// TIA Portal V20 export
TYPE "LConSMC_typeLineAxisActValues"
// Istwerte der Bahn / Actuak values of the web
// stored: Access Published
   STRUCT
      s : LReal;   // [m] / [ft] Position
      v : LReal;   // [m/min] / [ft/min] Geschwindigkeit / [m/min] / [ft/min] Velocity
   END_STRUCT;
END_TYPE
